// TIA Portal V17 export
// export: Created 2024-09-15T12:30:28.1842485Z, ExportSetting WithDefaults, DisplayName Totally Integrated Automation Portal, DisplayVersion V17, DisplayName TIA Portal Openness, DisplayVersion V17, DisplayName TIA Portal Version Control Interface, DisplayVersion V17, DisplayName STEP 7 Professional, DisplayVersion V17, DisplayName STEP 7 Safety, DisplayVersion V17, DisplayName WinCC Professional, DisplayVersion V17
TYPE "typ_Workpiece"
// stored: IsFailsafeCompliant false
   STRUCT
      s_id : String;   // Unique id of Workpiece
      s_type : String;   // Type of workpiece ("RED"/"WHITE"/"BLUE")
      s_state : String;   // State of workpiece ("RAW"/"PROCESSED"). Not really relevant since addind Workpiece_States
      Workpiece_States : "typ_Workpiece_States";   // Possible states of workpiece and timestamps
      Workpiece_Parameters : "typ_Workpiece_Parameters";   // Order parameters
   END_STRUCT;
END_TYPE
